{attribute 'linkalways'} 
{attribute 'no_explicit_call' := 'This FB is a CLASS and must be accessed using methods or properties'}
{attribute 'enable_dynamic_creation'}
FUNCTION_BLOCK _ETcVnBarcodeType EXTENDS EnumDatatypeBase
VAR
	localData : ETcVnBarcodeType;
	activeData : REFERENCE TO ETcVnBarcodeType;
	enumBaseDatatype : _UDINT(localData);
END_VAR

METHOD PRIVATE AddLocalEnumeration
VAR_INPUT
	Enumeration : T_MAXSTRING;
	Value : ETcVnBarcodeType;
END_VAR
AddEnumeration(Enumeration, Value);
END_METHOD

PROPERTY PUBLIC Address : PVOID
GET
Address := ADR(activeData);
END_GET
END_PROPERTY

METHOD PUBLIC ClearReference
VAR_INPUT
END_VAR
activeData REF= localData;
SetBaseDatatypeReference();
END_METHOD

METHOD PUBLIC Clone : I_Datatype
VAR
    pClone : POINTER TO _ETcVnBarcodeType;
END_VAR
pClone := __NEW(_ETcVnBarcodeType(InitialValue := Value));
Clone := pClone^;
END_METHOD

METHOD FB_init : BOOL
VAR_INPUT
	bInitRetains : BOOL; // if TRUE, the retain variables are initialized (warm start / cold start)
	bInCopyCode : BOOL;  // if TRUE, the instance afterwards gets moved into the copy code (online change)
	InitialValue : ETcVnBarcodeType;
END_VAR
localData := InitialValue;
AddBaseDatatype(enumBaseDatatype);
ClearReference();

AddLocalEnumeration('TCVN_BT_CODABAR', ETcVnBarcodeType.TCVN_BT_CODABAR);
AddLocalEnumeration('TCVN_BT_CODE39', ETcVnBarcodeType.TCVN_BT_CODE39);
AddLocalEnumeration('TCVN_BT_CODE93', ETcVnBarcodeType.TCVN_BT_CODE93);
AddLocalEnumeration('TCVN_BT_CODE128', ETcVnBarcodeType.TCVN_BT_CODE128);
AddLocalEnumeration('TCVN_BT_EAN8', ETcVnBarcodeType.TCVN_BT_EAN8);
AddLocalEnumeration('TCVN_BT_EAN13', ETcVnBarcodeType.TCVN_BT_EAN13);
AddLocalEnumeration('TCVN_BT_ITF', ETcVnBarcodeType.TCVN_BT_ITF);
AddLocalEnumeration('TCVN_BT_UPCA', ETcVnBarcodeType.TCVN_BT_UPCA);
AddLocalEnumeration('TCVN_BT_UPCE', ETcVnBarcodeType.TCVN_BT_UPCE);
AddLocalEnumeration('TCVN_BT_ANY', ETcVnBarcodeType.TCVN_BT_ANY);
AddLocalEnumeration('TCVN_BT_CODE39EXTENDED', ETcVnBarcodeType.TCVN_BT_CODE39EXTENDED);
END_METHOD

PROPERTY PUBLIC Identifier : T_MAXSTRING
GET
Identifier := 'ETcVnBarcodeType';
END_GET
END_PROPERTY

METHOD IsEnumeratorValueEqual : BOOL
VAR_INPUT
	Enumerator : I_KeyValueForwardEnumerator;
END_VAR
VAR
	storedValue : ETcVnBarcodeType;
END_VAR
IF NOT Enumerator.TryGet(storedValue) THEN
	RETURN;
END_IF

IsEnumeratorValueEqual := storedValue = activeData;
END_METHOD

METHOD PUBLIC MakeReferenceTo
VAR_INPUT
	ReferenceTarget : REFERENCE TO ETcVnBarcodeType;
END_VAR
activeData REF= ReferenceTarget;
SetBaseDatatypeReference();
END_METHOD

METHOD PROTECTED SetBaseDatatypeReference
VAR_INPUT
END_VAR
enumBaseDatatype.MakeReferenceTo(activeData);
END_METHOD

PROPERTY PUBLIC Size : UDINT
GET
Size := SIZEOF(activeData);
END_GET
END_PROPERTY

METHOD TryMakeReferenceTo : BOOL
VAR_INPUT
	Target : I_Datatype;
END_VAR
VAR
	pTargetData : POINTER TO ETcVnBarcodeType;
END_VAR
IF NOT IsEquivalentTo(Target) THEN
	RETURN;
END_IF

pTargetData := Target.Address;
activeData REF= pTargetData^;
SetBaseDatatypeReference();
TryMakeReferenceTo := TRUE;
END_METHOD

PROPERTY PUBLIC Value : ETcVnBarcodeType
GET
Value := activeData;
END_GET
SET
activeData := Value;
END_SET
END_PROPERTY

END_FUNCTION_BLOCK

(* stored: Version 1.1.0.1, ProductVersion 3.1.4024.13
   POU _ETcVnBarcodeType: Id {7a3e74bc-ac60-444c-92ad-a9f581cd30af}, SpecialFunc None
   Folder Core: Id {898d1d88-14b7-0eff-00f8-5c62e1f2f445}
   Folder Protected: Id {1387034a-b0fa-05b9-24a9-5edcd278ecf6}
   Folder Customize: Id {d13d5038-0f27-0fd6-27c9-29f195db7ed1}
   Folder Constructor: Id {f33d2166-2ee1-489a-b415-e146babb8ee2}
   Folder Private: Id {1316053d-d1f5-46b2-9db7-c78d9e73026a}
   Folder Protected: Id {07784be0-eda4-433f-a31d-9ffffb062de4}
   Method AddLocalEnumeration: Id {fc2bcb12-f417-4bee-ae26-0036007422f1}
   Property Address: Id {ec3fea57-451f-07f0-22fa-5f263e96675c}
   Get Get: Id {01993e8a-a8fd-0b65-1224-b6dcfd454f96}
   Method ClearReference: Id {88e044d9-a59c-06e5-3220-04fc667cb6bc}
   Method Clone: Id {cf0d44a2-0a15-4260-93c5-731ac9834afb}
   Method FB_init: Id {a4678cee-fbfd-418c-9b3c-3aff4f842516}
   Property Identifier: Id {d22256cd-c98c-486e-9fe4-d8801a3b7fd0}
   Get Get: Id {0c2dc1d3-9639-400e-a40e-f77764a61f6f}
   Method IsEnumeratorValueEqual: Id {62b17a6d-c020-42b0-8569-d9056dfde073}
   Method MakeReferenceTo: Id {4f8e3114-2194-4fcc-8b7d-936efc562493}
   Method SetBaseDatatypeReference: Id {cb249af7-9937-0fa1-1068-85e5a7230760}
   Property Size: Id {214cf22d-d626-0b14-20de-2d2697952e1c}
   Get Get: Id {ffb88735-af32-0d32-2d52-9d29bbc183b7}
   Method TryMakeReferenceTo: Id {8e1d0dd2-5f5f-4200-a9f1-d1d872ff3e82}
   Property Value: Id {65d59710-47eb-41ad-8288-452b4b5617d3}
   Get Get: Id {5910f5b0-24a4-4661-aaf3-166bb13f57a8}
   Set Set: Id {22736f2a-79f2-4b5e-9495-667987906689} *)
